// TIA Portal V17 export
// export: Created 2025-06-25T13:13:24.9076764Z, ExportSetting WithDefaults, DisplayName Totally Integrated Automation Portal, DisplayVersion V17 Update 8, DisplayName TIA Portal Openness, DisplayVersion V17 Update 8, DisplayName TIA Portal Version Control Interface, DisplayVersion V17, DisplayName STEP 7 Professional, DisplayVersion V17 Update 8, DisplayName STEP 7 Safety, DisplayVersion V17 Update 6, DisplayName WinCC Advanced, DisplayVersion V17 Update 8
DATA_BLOCK "DB_CurrentSetting"   // DB21
{ S7_Optimized_Access := 'TRUE' }
AUTHOR : AZ
VERSION : 0.1
// stored: AutoNumber true, DBAccessibleFromOPCUA true, DBAccessibleFromWebserver true, InstanceOfName CurrentSetting-STRUCT, InstanceOfType UDT, IsOnlyStoredInLoadMemory false, IsWriteProtectedInAS false
"CurrentSetting-STRUCT"
   // VAR RETAIN
   //    Fluid { S7_SetPoint := 'True'} : "FluidData-STRUCT";
   //    Compressor { S7_SetPoint := 'True'} : "CompressorData-STRUCT";
   //    System { S7_SetPoint := 'True'} : "SystemData-STRUCT";
   //    VariableSetting { S7_SetPoint := 'True'} : "VariableSetting-STRUCT";
   //    StaticSetting { S7_SetPoint := 'True'} : "StaticSetting-STRUCT";
   //    NewInitialisation_Required : Bool := FALSE;
   //    ParameterSet_Ordered : Bool := FALSE;
   //    ParameterSet_Indicator : Bool := FALSE;
   //    MissingSetting : Struct
   //       Compressor : Struct
   //          OilPumpCurveCritical : Real := 0.133;
   //          OilPumpCurveWarning : Real := 0.166;
   //          MinStartupSpeed : Real := 25.0;
   //          WarmupSpeed : Real := 550.0;
   //          MinOperationalSpeed : Real := 550.0;
   //          MaxOperationalSpeed : Real := 650.0;
   //          OilFilterDeltaPCritical : Real := 150.0;
   //          OilFilterDeltaPWarning : Real := 100.0;
   //       END_STRUCT;
   //       System : Struct
   //          HydrolockSpeed : Real := 330.0;
   //          CondenserCoefficient : Real := 13.024;
   //          EvaporatorCoefficient : Real := 19.07;
   //          SuctionLineDryLimitPressure : Real := 80.0;
   //          SuctionLineDryLimitSuperheat : Real := 27.0;
   //          CompressorSuperheatDischargeMinimum : Real := 20.0;
   //          RecuperatorDeltaTWorking : Real := 3.0;
   //          RecuperatorDeltaTNotWorking : Real := -2.0;
   //          ExpansionValvePositionStart : Real := 5.5;
   //          ExpansionValvePositionStartCold : Real := 3.0;
   //          HeatSourceDeltaPFlow : Real := 2.0;
   //          HeatSinkDeltaPFlow : Real := 2.0;
   //       END_STRUCT;
   //       Misc : Struct
   //          CompressorStoppedLimit : Real := 10.0;
   //          State2DwellTime { S7_SetPoint := 'True'} : Time := T#10S;
   //          State3DwellTime : Time := T#30S;
   //          State4DwellTime : Time := T#30S;
   //          State5DwellTime : Time := T#20M;
   //          State7DwellTime : Time := T#10S;
   //          State2PauseTime : Time := T#10S;
   //          EmergencyStopWaitTime : Time := T#5M;
   //          T_HeatSinkTemperatureIn_Max : Real := 75.0;
   //       END_STRUCT;
   //    END_STRUCT;
   // END_VAR
BEGIN
   Fluid."Name" := 'R1233zdE';
   Fluid.FluidTypeNumber := 2;
   Fluid.SaturationCurve_Temperature_C[0] := -10.0;
   Fluid.SaturationCurve_Temperature_C[1] := -5.4872;
   Fluid.SaturationCurve_Temperature_C[2] := -0.9744;
   Fluid.SaturationCurve_Temperature_C[3] := 3.5385;
   Fluid.SaturationCurve_Temperature_C[4] := 8.0513;
   Fluid.SaturationCurve_Temperature_C[5] := 12.5641;
   Fluid.SaturationCurve_Temperature_C[6] := 17.0769;
   Fluid.SaturationCurve_Temperature_C[7] := 21.5897;
   Fluid.SaturationCurve_Temperature_C[8] := 26.1026;
   Fluid.SaturationCurve_Temperature_C[9] := 30.6154;
   Fluid.SaturationCurve_Temperature_C[10] := 35.1282;
   Fluid.SaturationCurve_Temperature_C[11] := 39.641;
   Fluid.SaturationCurve_Temperature_C[12] := 44.1538;
   Fluid.SaturationCurve_Temperature_C[13] := 48.6667;
   Fluid.SaturationCurve_Temperature_C[14] := 53.1795;
   Fluid.SaturationCurve_Temperature_C[15] := 57.6923;
   Fluid.SaturationCurve_Temperature_C[16] := 62.2051;
   Fluid.SaturationCurve_Temperature_C[17] := 66.7179;
   Fluid.SaturationCurve_Temperature_C[18] := 71.2308;
   Fluid.SaturationCurve_Temperature_C[19] := 75.7436;
   Fluid.SaturationCurve_Temperature_C[20] := 80.2564;
   Fluid.SaturationCurve_Temperature_C[21] := 84.7692;
   Fluid.SaturationCurve_Temperature_C[22] := 89.2821;
   Fluid.SaturationCurve_Temperature_C[23] := 93.7949;
   Fluid.SaturationCurve_Temperature_C[24] := 98.3077;
   Fluid.SaturationCurve_Temperature_C[25] := 102.8205;
   Fluid.SaturationCurve_Temperature_C[26] := 107.3333;
   Fluid.SaturationCurve_Temperature_C[27] := 111.8462;
   Fluid.SaturationCurve_Temperature_C[28] := 116.359;
   Fluid.SaturationCurve_Temperature_C[29] := 120.8718;
   Fluid.SaturationCurve_Temperature_C[30] := 125.3846;
   Fluid.SaturationCurve_Temperature_C[31] := 129.8974;
   Fluid.SaturationCurve_Temperature_C[32] := 134.4103;
   Fluid.SaturationCurve_Temperature_C[33] := 138.9231;
   Fluid.SaturationCurve_Temperature_C[34] := 143.4359;
   Fluid.SaturationCurve_Temperature_C[35] := 147.9487;
   Fluid.SaturationCurve_Temperature_C[36] := 152.4615;
   Fluid.SaturationCurve_Temperature_C[37] := 156.9744;
   Fluid.SaturationCurve_Temperature_C[38] := 161.4872;
   Fluid.SaturationCurve_Temperature_C[39] := 166.0;
   Fluid.SaturationCurve_Temperature_C[40] := 172.9092;
   Fluid.SaturationCurve_Pressure_kPa[0] := 30.3567;
   Fluid.SaturationCurve_Pressure_kPa[1] := 37.5596;
   Fluid.SaturationCurve_Pressure_kPa[2] := 46.0817;
   Fluid.SaturationCurve_Pressure_kPa[3] := 56.0903;
   Fluid.SaturationCurve_Pressure_kPa[4] := 67.7633;
   Fluid.SaturationCurve_Pressure_kPa[5] := 81.2888;
   Fluid.SaturationCurve_Pressure_kPa[6] := 96.865;
   Fluid.SaturationCurve_Pressure_kPa[7] := 114.6997;
   Fluid.SaturationCurve_Pressure_kPa[8] := 135.0095;
   Fluid.SaturationCurve_Pressure_kPa[9] := 158.0203;
   Fluid.SaturationCurve_Pressure_kPa[10] := 183.9659;
   Fluid.SaturationCurve_Pressure_kPa[11] := 213.0886;
   Fluid.SaturationCurve_Pressure_kPa[12] := 245.6381;
   Fluid.SaturationCurve_Pressure_kPa[13] := 281.8717;
   Fluid.SaturationCurve_Pressure_kPa[14] := 322.0539;
   Fluid.SaturationCurve_Pressure_kPa[15] := 366.4563;
   Fluid.SaturationCurve_Pressure_kPa[16] := 415.3576;
   Fluid.SaturationCurve_Pressure_kPa[17] := 469.0435;
   Fluid.SaturationCurve_Pressure_kPa[18] := 527.8071;
   Fluid.SaturationCurve_Pressure_kPa[19] := 591.9489;
   Fluid.SaturationCurve_Pressure_kPa[20] := 661.7775;
   Fluid.SaturationCurve_Pressure_kPa[21] := 737.6098;
   Fluid.SaturationCurve_Pressure_kPa[22] := 819.7723;
   Fluid.SaturationCurve_Pressure_kPa[23] := 908.6015;
   Fluid.SaturationCurve_Pressure_kPa[24] := 1004.446;
   Fluid.SaturationCurve_Pressure_kPa[25] := 1107.666;
   Fluid.SaturationCurve_Pressure_kPa[26] := 1218.639;
   Fluid.SaturationCurve_Pressure_kPa[27] := 1337.757;
   Fluid.SaturationCurve_Pressure_kPa[28] := 1465.436;
   Fluid.SaturationCurve_Pressure_kPa[29] := 1602.111;
   Fluid.SaturationCurve_Pressure_kPa[30] := 1748.251;
   Fluid.SaturationCurve_Pressure_kPa[31] := 1904.356;
   Fluid.SaturationCurve_Pressure_kPa[32] := 2070.969;
   Fluid.SaturationCurve_Pressure_kPa[33] := 2248.688;
   Fluid.SaturationCurve_Pressure_kPa[34] := 2438.177;
   Fluid.SaturationCurve_Pressure_kPa[35] := 2640.193;
   Fluid.SaturationCurve_Pressure_kPa[36] := 2855.623;
   Fluid.SaturationCurve_Pressure_kPa[37] := 3085.555;
   Fluid.SaturationCurve_Pressure_kPa[38] := 3331.466;
   Fluid.SaturationCurve_Pressure_kPa[39] := 3595.998;
   Fluid.SaturationCurve_Pressure_kPa[40] := 4001.0;
   Fluid.DensityCurve_Pressure_kPa[0] := 50.0;
   Fluid.DensityCurve_Pressure_kPa[1] := 74.7475;
   Fluid.DensityCurve_Pressure_kPa[2] := 173.05;
   Fluid.DensityCurve_Pressure_kPa[3] := 388.0866;
   Fluid.DensityCurve_Pressure_kPa[4] := 746.4811;
   Fluid.DensityCurve_Pressure_kPa[5] := 1244.251;
   Fluid.DensityCurve_Pressure_kPa[6] := 1836.598;
   Fluid.DensityCurve_Pressure_kPa[7] := 2441.284;
   Fluid.DensityCurve_Pressure_kPa[8] := 2962.33;
   Fluid.DensityCurve_Pressure_kPa[9] := 3328.69;
   Fluid.DensityCurve_Pressure_kPa[10] := 3526.57;
   Fluid.DensityCurve_Pressure_kPa[11] := 3613.637;
   Fluid.DensityCurve_Pressure_kPa[12] := 4001.0;
   Fluid.DensityCurveLiquide_Densety_kg_m3[0] := 1319.278;
   Fluid.DensityCurveLiquide_Densety_kg_m3[1] := 1297.254;
   Fluid.DensityCurveLiquide_Densety_kg_m3[2] := 1242.459;
   Fluid.DensityCurveLiquide_Densety_kg_m3[3] := 1173.489;
   Fluid.DensityCurveLiquide_Densety_kg_m3[4] := 1098.545;
   Fluid.DensityCurveLiquide_Densety_kg_m3[5] := 1019.4;
   Fluid.DensityCurveLiquide_Densety_kg_m3[6] := 936.68;
   Fluid.DensityCurveLiquide_Densety_kg_m3[7] := 851.4562;
   Fluid.DensityCurveLiquide_Densety_kg_m3[8] := 765.7374;
   Fluid.DensityCurveLiquide_Densety_kg_m3[9] := 682.3312;
   Fluid.DensityCurveLiquide_Densety_kg_m3[10] := 605.4245;
   Fluid.DensityCurveLiquide_Densety_kg_m3[11] := 523.5075;
   Fluid.DensityCurveLiquide_Densety_kg_m3[12] := 455.9911;
   Fluid.DensityCurveVapor_Densety_kg_m3[0] := 2.9405;
   Fluid.DensityCurveVapor_Densety_kg_m3[1] := 4.2862;
   Fluid.DensityCurveVapor_Densety_kg_m3[2] := 9.4624;
   Fluid.DensityCurveVapor_Densety_kg_m3[3] := 20.5809;
   Fluid.DensityCurveVapor_Densety_kg_m3[4] := 39.5976;
   Fluid.DensityCurveVapor_Densety_kg_m3[5] := 68.316;
   Fluid.DensityCurveVapor_Densety_kg_m3[6] := 108.1358;
   Fluid.DensityCurveVapor_Densety_kg_m3[7] := 159.5525;
   Fluid.DensityCurveVapor_Densety_kg_m3[8] := 221.352;
   Fluid.DensityCurveVapor_Densety_kg_m3[9] := 289.9457;
   Fluid.DensityCurveVapor_Densety_kg_m3[10] := 359.0497;
   Fluid.DensityCurveVapor_Densety_kg_m3[11] := 437.3655;
   Fluid.DensityCurveVapor_Densety_kg_m3[12] := 455.9911;
   Fluid.DensityCurveVapor_SuperheatCorrection_a := 0.0;
   Fluid.DensityCurveVapor_SuperheatCorrection_b := 0.0002;
   Fluid.EnthalpyMap_Superheat_C[0] := -20.0;
   Fluid.EnthalpyMap_Superheat_C[1] := -6.0;
   Fluid.EnthalpyMap_Superheat_C[2] := -2.0;
   Fluid.EnthalpyMap_Superheat_C[3] := -0.01;
   Fluid.EnthalpyMap_Superheat_C[4] := 0.01;
   Fluid.EnthalpyMap_Superheat_C[5] := 2.0;
   Fluid.EnthalpyMap_Superheat_C[6] := 6.0;
   Fluid.EnthalpyMap_Superheat_C[7] := 18.0;
   Fluid.EnthalpyMap_Superheat_C[8] := 40.0;
   Fluid.EnthalpyMap_Pressure_kPa[0] := 100.0;
   Fluid.EnthalpyMap_Pressure_kPa[1] := 127.0833;
   Fluid.EnthalpyMap_Pressure_kPa[2] := 234.6644;
   Fluid.EnthalpyMap_Pressure_kPa[3] := 469.9978;
   Fluid.EnthalpyMap_Pressure_kPa[4] := 862.2203;
   Fluid.EnthalpyMap_Pressure_kPa[5] := 1406.974;
   Fluid.EnthalpyMap_Pressure_kPa[6] := 2055.23;
   Fluid.EnthalpyMap_Pressure_kPa[7] := 2716.992;
   Fluid.EnthalpyMap_Pressure_kPa[8] := 3287.218;
   Fluid.EnthalpyMap_Pressure_kPa[9] := 3688.158;
   Fluid.EnthalpyMap_Pressure_kPa[10] := 3904.715;
   Fluid.EnthalpyMap_Pressure_kPa[11] := 4000.0;
   Fluid.EnthalpyMap_Enthalpy_kJ_kg[0,0] := 197.5698;
   Fluid.EnthalpyMap_Enthalpy_kJ_kg[0,1] := 214.1515;
   Fluid.EnthalpyMap_Enthalpy_kJ_kg[0,2] := 218.9438;
   Fluid.EnthalpyMap_Enthalpy_kJ_kg[0,3] := 221.3373;
   Fluid.EnthalpyMap_Enthalpy_kJ_kg[0,4] := 416.1527;
   Fluid.EnthalpyMap_Enthalpy_kJ_kg[0,5] := 417.767;
   Fluid.EnthalpyMap_Enthalpy_kJ_kg[0,6] := 421.028;
   Fluid.EnthalpyMap_Enthalpy_kJ_kg[0,7] := 430.9391;
   Fluid.EnthalpyMap_Enthalpy_kJ_kg[0,8] := 449.5907;
   Fluid.EnthalpyMap_Enthalpy_kJ_kg[1,0] := 205.2355;
   Fluid.EnthalpyMap_Enthalpy_kJ_kg[1,1] := 221.9542;
   Fluid.EnthalpyMap_Enthalpy_kJ_kg[1,2] := 226.7875;
   Fluid.EnthalpyMap_Enthalpy_kJ_kg[1,3] := 229.2018;
   Fluid.EnthalpyMap_Enthalpy_kJ_kg[1,4] := 420.6821;
   Fluid.EnthalpyMap_Enthalpy_kJ_kg[1,5] := 422.3276;
   Fluid.EnthalpyMap_Enthalpy_kJ_kg[1,6] := 425.6502;
   Fluid.EnthalpyMap_Enthalpy_kJ_kg[1,7] := 435.7365;
   Fluid.EnthalpyMap_Enthalpy_kJ_kg[1,8] := 454.6786;
   Fluid.EnthalpyMap_Enthalpy_kJ_kg[2,0] := 227.161;
   Fluid.EnthalpyMap_Enthalpy_kJ_kg[2,1] := 244.2909;
   Fluid.EnthalpyMap_Enthalpy_kJ_kg[2,2] := 249.2492;
   Fluid.EnthalpyMap_Enthalpy_kJ_kg[2,3] := 251.7272;
   Fluid.EnthalpyMap_Enthalpy_kJ_kg[2,4] := 433.2917;
   Fluid.EnthalpyMap_Enthalpy_kJ_kg[2,5] := 435.0327;
   Fluid.EnthalpyMap_Enthalpy_kJ_kg[2,6] := 438.5429;
   Fluid.EnthalpyMap_Enthalpy_kJ_kg[2,7] := 449.1592;
   Fluid.EnthalpyMap_Enthalpy_kJ_kg[2,8] := 468.9681;
   Fluid.EnthalpyMap_Enthalpy_kJ_kg[3,0] := 256.9384;
   Fluid.EnthalpyMap_Enthalpy_kJ_kg[3,1] := 274.7034;
   Fluid.EnthalpyMap_Enthalpy_kJ_kg[3,2] := 279.8614;
   Fluid.EnthalpyMap_Enthalpy_kJ_kg[3,3] := 282.4424;
   Fluid.EnthalpyMap_Enthalpy_kJ_kg[3,4] := 449.3674;
   Fluid.EnthalpyMap_Enthalpy_kJ_kg[3,5] := 451.2598;
   Fluid.EnthalpyMap_Enthalpy_kJ_kg[3,6] := 455.0643;
   Fluid.EnthalpyMap_Enthalpy_kJ_kg[3,7] := 466.4958;
   Fluid.EnthalpyMap_Enthalpy_kJ_kg[3,8] := 487.595;
   Fluid.EnthalpyMap_Enthalpy_kJ_kg[4,0] := 288.6115;
   Fluid.EnthalpyMap_Enthalpy_kJ_kg[4,1] := 307.2277;
   Fluid.EnthalpyMap_Enthalpy_kJ_kg[4,2] := 312.6681;
   Fluid.EnthalpyMap_Enthalpy_kJ_kg[4,3] := 315.398;
   Fluid.EnthalpyMap_Enthalpy_kJ_kg[4,4] := 464.6608;
   Fluid.EnthalpyMap_Enthalpy_kJ_kg[4,5] := 466.762;
   Fluid.EnthalpyMap_Enthalpy_kJ_kg[4,6] := 470.9658;
   Fluid.EnthalpyMap_Enthalpy_kJ_kg[4,7] := 483.4603;
   Fluid.EnthalpyMap_Enthalpy_kJ_kg[4,8] := 506.1447;
   Fluid.EnthalpyMap_Enthalpy_kJ_kg[5,0] := 319.2484;
   Fluid.EnthalpyMap_Enthalpy_kJ_kg[5,1] := 339.0134;
   Fluid.EnthalpyMap_Enthalpy_kJ_kg[5,2] := 344.8686;
   Fluid.EnthalpyMap_Enthalpy_kJ_kg[5,3] := 347.8254;
   Fluid.EnthalpyMap_Enthalpy_kJ_kg[5,4] := 476.8875;
   Fluid.EnthalpyMap_Enthalpy_kJ_kg[5,5] := 479.2968;
   Fluid.EnthalpyMap_Enthalpy_kJ_kg[5,6] := 484.0675;
   Fluid.EnthalpyMap_Enthalpy_kJ_kg[5,7] := 497.9603;
   Fluid.EnthalpyMap_Enthalpy_kJ_kg[5,8] := 522.524;
   Fluid.EnthalpyMap_Enthalpy_kJ_kg[6,0] := 346.9259;
   Fluid.EnthalpyMap_Enthalpy_kJ_kg[6,1] := 368.272;
   Fluid.EnthalpyMap_Enthalpy_kJ_kg[6,2] := 374.7868;
   Fluid.EnthalpyMap_Enthalpy_kJ_kg[6,3] := 378.132;
   Fluid.EnthalpyMap_Enthalpy_kJ_kg[6,4] := 484.4899;
   Fluid.EnthalpyMap_Enthalpy_kJ_kg[6,5] := 487.4372;
   Fluid.EnthalpyMap_Enthalpy_kJ_kg[6,6] := 493.119;
   Fluid.EnthalpyMap_Enthalpy_kJ_kg[6,7] := 508.9522;
   Fluid.EnthalpyMap_Enthalpy_kJ_kg[6,8] := 535.7144;
   Fluid.EnthalpyMap_Enthalpy_kJ_kg[7,0] := 369.9632;
   Fluid.EnthalpyMap_Enthalpy_kJ_kg[7,1] := 393.4236;
   Fluid.EnthalpyMap_Enthalpy_kJ_kg[7,2] := 401.0829;
   Fluid.EnthalpyMap_Enthalpy_kJ_kg[7,3] := 405.235;
   Fluid.EnthalpyMap_Enthalpy_kJ_kg[7,4] := 486.2374;
   Fluid.EnthalpyMap_Enthalpy_kJ_kg[7,5] := 490.3629;
   Fluid.EnthalpyMap_Enthalpy_kJ_kg[7,6] := 497.6848;
   Fluid.EnthalpyMap_Enthalpy_kJ_kg[7,7] := 516.2058;
   Fluid.EnthalpyMap_Enthalpy_kJ_kg[7,8] := 545.3667;
   Fluid.EnthalpyMap_Enthalpy_kJ_kg[8,0] := 387.0381;
   Fluid.EnthalpyMap_Enthalpy_kJ_kg[8,1] := 412.9451;
   Fluid.EnthalpyMap_Enthalpy_kJ_kg[8,2] := 422.6469;
   Fluid.EnthalpyMap_Enthalpy_kJ_kg[8,3] := 429.1883;
   Fluid.EnthalpyMap_Enthalpy_kJ_kg[8,4] := 480.7851;
   Fluid.EnthalpyMap_Enthalpy_kJ_kg[8,5] := 488.3624;
   Fluid.EnthalpyMap_Enthalpy_kJ_kg[8,6] := 498.5881;
   Fluid.EnthalpyMap_Enthalpy_kJ_kg[8,7] := 520.3678;
   Fluid.EnthalpyMap_Enthalpy_kJ_kg[8,8] := 551.7377;
   Fluid.EnthalpyMap_Enthalpy_kJ_kg[9,0] := 397.8677;
   Fluid.EnthalpyMap_Enthalpy_kJ_kg[9,1] := 425.8558;
   Fluid.EnthalpyMap_Enthalpy_kJ_kg[9,2] := 438.3909;
   Fluid.EnthalpyMap_Enthalpy_kJ_kg[9,3] := 462.7447;
   Fluid.EnthalpyMap_Enthalpy_kJ_kg[9,4] := 463.5576;
   Fluid.EnthalpyMap_Enthalpy_kJ_kg[9,5] := 484.1742;
   Fluid.EnthalpyMap_Enthalpy_kJ_kg[9,6] := 497.9508;
   Fluid.EnthalpyMap_Enthalpy_kJ_kg[9,7] := 522.3931;
   Fluid.EnthalpyMap_Enthalpy_kJ_kg[9,8] := 555.3659;
   Fluid.EnthalpyMap_Enthalpy_kJ_kg[10,0] := 403.7939;
   Fluid.EnthalpyMap_Enthalpy_kJ_kg[10,1] := 433.1682;
   Fluid.EnthalpyMap_Enthalpy_kJ_kg[10,2] := 448.1372;
   Fluid.EnthalpyMap_Enthalpy_kJ_kg[10,3] := 467.0842;
   Fluid.EnthalpyMap_Enthalpy_kJ_kg[10,4] := 467.3177;
   Fluid.EnthalpyMap_Enthalpy_kJ_kg[10,5] := 483.0886;
   Fluid.EnthalpyMap_Enthalpy_kJ_kg[10,6] := 498.0977;
   Fluid.EnthalpyMap_Enthalpy_kJ_kg[10,7] := 523.751;
   Fluid.EnthalpyMap_Enthalpy_kJ_kg[10,8] := 557.4834;
   Fluid.EnthalpyMap_Enthalpy_kJ_kg[11,0] := 406.426;
   Fluid.EnthalpyMap_Enthalpy_kJ_kg[11,1] := 436.4671;
   Fluid.EnthalpyMap_Enthalpy_kJ_kg[11,2] := 452.4549;
   Fluid.EnthalpyMap_Enthalpy_kJ_kg[11,3] := 469.0933;
   Fluid.EnthalpyMap_Enthalpy_kJ_kg[11,4] := 469.2745;
   Fluid.EnthalpyMap_Enthalpy_kJ_kg[11,5] := 483.1994;
   Fluid.EnthalpyMap_Enthalpy_kJ_kg[11,6] := 498.3468;
   Fluid.EnthalpyMap_Enthalpy_kJ_kg[11,7] := 524.4174;
   Fluid.EnthalpyMap_Enthalpy_kJ_kg[11,8] := 558.4523;
   Fluid.Limits.T_HeatSourceTemperature_Max := 120.0;
   Fluid.Limits.T_HeatSourceTemperature_Min := 55.0;
   Fluid.Limits.T_HeatSinkTemperature_Max := 150.0;
   Fluid.Limits.T_OilTemperature_Critical := 140.0;
   Fluid.Limits.T_OilSuperheat := 15.0;
   Fluid.Limits.T_CoolingSetpoint := 0.0;
   Fluid.T_AdditionalSuperHeatEvaporator := 8.0;
   Fluid.P_CriticalPoint := 3623.637;
   Compressor.CompressorTypeNumber := 1;
   Compressor.Limits.p_CrankCase_Max := 1600.0;
   Compressor.Limits.p_Oil_Min := 30.0;
   Compressor.Limits.n_Compressor_Max := 1200.0;
   Compressor.Limits.T_Motor_Max := 90.0;
   Compressor.Limits.M_Motor_Limit := 61.4;
   Compressor.Limits.T_Inverter_Max := 60.0;
   Compressor.Constant.CompressionVolume_L := 16.4;
   Compressor.Constant.CompressionLostPerPressureRatio := 3.41;
   Compressor.Constant.PumpEfficinecy := 93.69;
   Compressor.Settings := FALSE;
   System.SystemTypeNumber := 2;
   System.Limits.T_SuperHeatCompressorIn_Min := 2.0;
   System.Limits.T_Housing_Max := 50.0;
   System.Limits.T_CoolingCycle_Max := 65.0;
   System.Limits.p_CompressorOut_Max := 2700.0;
   System.Limits.p_EvaporatorOut_Max := 1550.0;
   System.Constant := FALSE;
   System.Settings.CooliungPump_ReversedPWM := FALSE;
   System.Settings.MotorCooling_AirFanCooledCycle := FALSE;
   System.Settings.DoubleExpansionValves := TRUE;
   System.Settings.Reserve3 := FALSE;
   System.Settings.Reserve4 := FALSE;
   System.Settings.Reserve5 := FALSE;
   VariableSetting.SystemType := 2;   // 1 = Alpha-1, 2 = Alpha-2
   VariableSetting.CompressorType := 1;
   VariableSetting.FluidType := 2;
   VariableSetting.OilPreheating_acv := TRUE;
   VariableSetting.OilHeatSetpoint_min := 45.0;
   VariableSetting.EnableViaHMI := TRUE;
   VariableSetting.EnableViaApplication := TRUE;
   VariableSetting.SourceOkFromApplication := FALSE;
   VariableSetting.SinkOkFromApplication := FALSE;
   VariableSetting.HeatSourceExternalControl := TRUE;
   VariableSetting.HeatSinkExternalControl := TRUE;
   StaticSetting.AdditionalSuperHeatOnColdStart := 0.0;
   StaticSetting.Limits.T_Ambient_Max := 40.0;
   StaticSetting.Limits.T_Cabinet_Max := 45.0;
END_DATA_BLOCK
